PROGRAM MAIN
VAR
END_VAR

END_PROGRAM

(* stored: Version 1.1.0.1
   POU MAIN: Id {b60edc56-17cb-40ee-9368-4c077c445fa6} *)
